{attribute 'GeneratedUsingTerminal: EJ5151-0000-0016'}
{attribute addProperty BoxType "EJ5151-0000-0016"}
{attribute addProperty Id "StatusAT %I*Status_3E6F3FF310Counter_valueAT %I*UINT2Latch_valueAT %I*UINT2"}
{attribute addProperty CRC "3008586885"}
{attribute addProperty Size "14"}
TYPE ENC_Inputs_B3536485 EXTENDS InputBase_8311D824 :
STRUCT
	{attribute addProperty Name "Status"}
	Status AT %I* : Status_3E6F3FF3;
	{attribute addProperty Name "Counter_value"}
	Counter_value AT %I* : UINT;
	{attribute addProperty Name "Latch_value"}
	Latch_value AT %I* : UINT;
END_STRUCT
END_TYPE

(* stored: Version 1.2.0.0, ProductVersion 3.1.4024.9
   DUT ENC_Inputs_B3536485: Id {aa11c87d-4332-46cc-a32d-676e1b290b6b} *)
